Fanuc KAREL source: compact_preamble.KL

PROGRAM KT00344
%NOLOCKGROUP
VAR
H1 : ARRAY[2] OF SHORT
R2:REAL
OUT:BOOLEAN
BEGIN
H1[1]=2
R2=3.0
OUT=((H1[1]) < R2)
END KT00344
